(* IEC 61131-3 sources: eCockpitGit/test_project/src/%F%00 Library/%F%Common Functions/%F%Dynamic Array/%POU%FB_wDynamicSortedArray, 6 files *)

(* ---- %METH%addElement.st ---- *)
//NON-Blocking method, is not threadsafe without calling getExclusive access before use
//Appends element to array
// |**Version**|**Author**| **Date** |**Changes**
// | 1         | NSN      | 18-05-22 | Creation
METHOD addElement : SLMResult
VAR_INPUT
	element			:WORD;	//Element to append
END_VAR
VAR_OUTPUT
	index			:WORD;
END_VAR
VAR
	i				:WORD;
	size			:WORD;		//Size to allocate to array
	offset			:WORD;
	newArrayBuffer	:POINTER TO ARRAY[0..99] OF WORD;
END_VAR

(*%!%__DELIMITER__%!%*)
IF S_lenght < S_maxSize THEN
	IF S_map THEN
		IF checkExists(element:=element) THEN
			addElement.success			:=		FALSE;
			addElement.code				:=		ERCodes.FB_DynamicArray_addElement;
			addElement.reason			:=		GTErrors.EelementInArray;
			RETURN;
		END_IF
	END_IF
	//If array is full, then more space is allocated
	IF S_lenght < S_blockSize THEN
		FOR i := S_lenght TO 1 BY -1 DO
			IF S_array^[i - 1] <= element THEN
				S_array^[i]				:=		element;
				EXIT;
			ELSE
				S_array^[i]				:=		S_array^[i - 1];
			END_IF
		END_FOR
		IF i = 0 THEN
			S_array^[0]					:=		element;
		END_IF
	ELSE
		//Size is corrected to increment size
		size								:=		((S_blockSize / S_increment) + 1) * S_increment;
		//Byte size is calculated
		newArrayBuffer						:=		__NEW(WORD,size);
		//If the memory manager fails, the registerering fails
		IF newArrayBuffer = 0 THEN
			addElement.success				:=		FALSE;
			addElement.code					:=		ERCodes.FB_DynamicArray_allocateInternal;
			addElement.reason				:=		GTErrors.EoutOfDynamicMemory;
			RETURN;
		END_IF
		//The contens of the old buffer is copied to the new buffer
		IF S_lenght > 0 THEN
			FOR i := 0 TO S_lenght - 1 DO
				IF offset = 0 AND S_array^[i] >= element THEN
					newArrayBuffer^[i]		:=		element;
					offset					:=		1;
				END_IF
				newArrayBuffer^[i + offset]	:=		S_array^[i];
			END_FOR
			IF offset = 0 AND i = S_lenght THEN
				newArrayBuffer^[i]			:=		element;
			END_IF
		ELSE
			newArrayBuffer^[0]				:=		element;
		END_IF
		//Old array memory is deleted, and new one is use
		FU_SafeDelete(pMem:=S_array);
		S_array								:=		newArrayBuffer;
		S_blockSize							:=		size;
	END_IF
	index									:=		S_lenght;
	S_lenght								:=		S_lenght + 1;
ELSE
	addElement.success						:=		FALSE;
	addElement.code							:=		ERCodes.FB_DynamicArray_addElement;
	addElement.reason						:=		GTErrors.EarrayFull;
END_IF

(* ---- %METH%allocate.st ---- *)
//NON-Blocking method, is not threadsafe without calling getExclusive access before use
//Pre-allocates a given size to the array
// |**Version**|**Author**| **Date** |**Changes**
// | 1         | NSN      | 18-05-22 | Creation
METHOD allocate :SLMResult
VAR_INPUT
	size			:WORD;		//Size to allocate to array
END_VAR
VAR
	newArrayBuffer	:POINTER TO ARRAY[0..99] OF WORD;
END_VAR
(*%!%__DELIMITER__%!%*)
IF size > S_blockSize THEN
	//Size is corrected to increment size
	size							:=		(((size - 1) / S_increment) + 1) * S_increment;
	//Byte size is calculated
	newArrayBuffer					:=		__NEW(WORD,size);
	//If the memory manager fails, the registerering fails
	IF newArrayBuffer = 0 THEN
		allocate.success			:=		FALSE;
		allocate.code				:=		ERCodes.FB_DynamicArray_allocateInternal;
		allocate.reason				:=		GTErrors.EoutOfDynamicMemory;
		RETURN;
	END_IF
	//The contens of the old buffer is copied to the new buffer
	IF S_lenght > 0 THEN
		SysMem.SysMemCpy(pDest:=newArrayBuffer,pSrc:=S_array,udiCount:=S_lenght * 2);
	END_IF
	//Old array memory is deleted, and new one is use
	FU_SafeDelete(pMem:=S_array);
	S_array							:=		newArrayBuffer;
	S_blockSize						:=		size;
END_IF

(* ---- %METH%checkExists.st ---- *)
//NON-Blocking method, is not threadsafe without calling getExclusive access before use
//Checks if element exist in array, and returns index of element in array
//Returns true if element is found
// |**Version**|**Author**| **Date** |**Changes**
// | 1         | NSN      | 18-05-22 | Creation
METHOD checkExists : BOOL
VAR_INPUT
	element		:WORD;		//Element to check
END_VAR
VAR_OUTPUT
	index		:WORD;		//Index of found element
END_VAR
VAR
	lower		:DINT;
	upper		:DINT := S_lenght - 1;
END_VAR
(*%!%__DELIMITER__%!%*)
IF S_lenght > 0 THEN
	WHILE TRUE DO
		index					:=		 TO_WORD(SHR((lower + upper),1));
		IF S_array^[index] > element THEN
			upper				:=		index - 1;
		ELSIF S_array^[index] < element THEN
			lower				:=		index + 1;
		ELSE
			checkExists			:=		TRUE;
			RETURN;
		END_IF
		IF lower > upper THEN
			index				:=		0;
			RETURN;
		END_IF
	END_WHILE
END_IF

(* ---- %METH%getElementByIndex.st ---- *)
//Returns the element at the given index
// |**Version**|**Author**| **Date** |**Changes**
// | 1         | NSN      | 18-05-22 | Creation
METHOD getElementByIndex : SLMResult
VAR_INPUT
	index			:WORD;
END_VAR
VAR_OUTPUT
	element			:WORD;
END_VAR
(*%!%__DELIMITER__%!%*)
IF index < S_lenght THEN
	element								:=		S_array^[index];
ELSE
	getElementByIndex.success		:=		FALSE;
	getElementByIndex.code			:=		ERCodes.FB_DynamicArray_removeElementByIndex;
	getElementByIndex.reason		:=		GTErrors.EindexOutOfRange;
END_IF

(* ---- %METH%removeElement.st ---- *)
//NON-Blocking method, is not threadsafe without calling getExclusive access before use
//Finds and removes the given element from the array, if multiple are found the amount of elements removed are limited by the amount given
// |**Version**|**Author**| **Date** |**Changes**
// | 1         | NSN      | 18-05-22 | Creation
METHOD removeElement
VAR_INPUT
	element			:WORD;		//Element to remove
	amount			:WORD;		//Max amount of same elements to remove from array, 0 means all
END_VAR
VAR
	i				:WORD;
	offset			:WORD;
END_VAR
(*%!%__DELIMITER__%!%*)
IF S_lenght > 0 THEN
	FOR i := 0 TO S_lenght - 1 DO
		IF S_array^[i] = element AND (offset < amount OR amount = 0) THEN
			offset					:=		offset + 1;
		ELSIF offset > 0 THEN
			S_array^[i - offset]	:=		S_array^[i];
		END_IF
	END_FOR
	S_lenght						:=		S_lenght - offset;
	IF S_lenght = 0 THEN
		S_blockSize					:=		0;
		FU_SafeDelete(pMem:=S_array);
	END_IF
END_IF

(* ---- %METH%removeElementByIndex.st ---- *)
//NON-Blocking method, is not threadsafe without calling getExclusive access before use
//Removes a given index from the array, by shifting all memory after it over it
// |**Version**|**Author**| **Date** |**Changes**
// | 1         | NSN      | 18-05-22 | Creation
METHOD removeElementByIndex : SLMResult
VAR_INPUT
	index			:WORD;		//Index to remove element from
END_VAR

(*%!%__DELIMITER__%!%*)
IF index < S_lenght THEN
	S_lenght							:=		S_lenght - 1;
	SysMem.SysMemCpy(pDest:=S_array + (index * 2),pSrc:=S_array + ((index + 1) * 2),udiCount:=(S_lenght - index) * 2);
	IF S_lenght = 0 THEN
		S_blockSize						:=		0;
		FU_SafeDelete(pMem:=S_array);
	END_IF
ELSE
	removeElementByIndex.success		:=		FALSE;
	removeElementByIndex.code			:=		ERCodes.FB_DynamicArray_removeElementByIndex;
	removeElementByIndex.reason			:=		GTErrors.EindexOutOfRange;
END_IF
